Staubli VAL3: actGesture.pgx

program actGesture()
begin
  putln("GestureCalled")
  putln(sInput)
  if (sInput == "fist")
    call gestureFist()
  endIf

end
